FUNCTION cot : lreal
VAR_INPUT
	i_angle:LREAL;
END_VAR
VAR
END_VAR

cot:=COS(i_angle)/SIN(i_angle);

END_FUNCTION

(* stored: Version 1.1.0.1, ProductVersion 3.1.4024.12
   POU cot: Id {b1447afa-f0f1-4b0a-b52c-db57e7ce69c7}, SpecialFunc None *)
